{attribute addProperty BoxType "ELM3002-0000-0016"}
{attribute addProperty Id "SamplesAT %I*ARRAY [0..0] OF DINT324"}
{attribute addProperty CRC "1340537356"}
{attribute addProperty SizeInBites "32"}
{attribute addProperty SizeInBytes "4"}
TYPE PAI_Samples_1_Channel_4FE6FA0C :
STRUCT
	{attribute addProperty Name "Samples"}
	Samples AT %I* : ARRAY [0..0] OF DINT;
END_STRUCT
END_TYPE

(* stored: Version 1.2.0.0, ProductVersion 3.1.4024.9
   DUT PAI_Samples_1_Channel_4FE6FA0C: Id {cbfca74b-7835-4245-a635-44a113eb113e} *)
